// TIA Portal V16 export
// export: Created 2022-11-14T17:35:22.3849211Z, ExportSetting WithDefaults, DisplayName Totally Integrated Automation Portal, DisplayVersion V16, DisplayName TIA Portal Version Control Interface, DisplayVersion V16, DisplayName TIA Portal Openness, DisplayVersion V16, DisplayName STEP 7 Professional, DisplayVersion V16, DisplayName STEP 7 Safety, DisplayVersion V16, DisplayName WinCC Advanced, DisplayVersion V16
FUNCTION "Denormalisation" : Void   // FC14, FBD
{ S7_Optimized_Access := 'TRUE' }
VERSION : 0.1
// stored: AutoNumber true, IsIECCheckEnabled false, SetENOAutomatically false, UDAEnableTagReadback false
   VAR_INPUT
      actual_value_INT : Int;
      normalisation : Real;
   END_VAR
   VAR_OUTPUT
      actual_value_REAL : Real;
   END_VAR
   VAR_TEMP
      temp_actual_value_DINT : DInt;
      temp_actual_value_REAL : Real;
   END_VAR
BEGIN

REGION Network 1
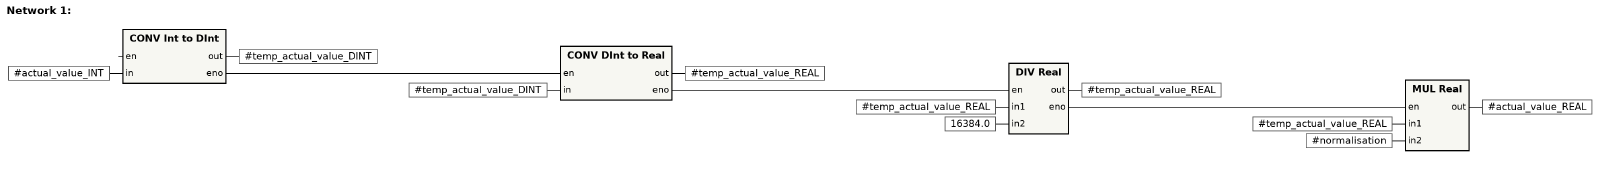
   // ENO of a box is taken as its EN; it also drops when the box reports an error
   #temp_actual_value_DINT := INT_TO_DINT(#actual_value_INT);
   #temp_actual_value_REAL := DINT_TO_REAL(#temp_actual_value_DINT);
   #temp_actual_value_REAL := #temp_actual_value_REAL / 16384.0;
   #actual_value_REAL := #temp_actual_value_REAL * #normalisation;
END_REGION
END_FUNCTION
